TYPE ST_IoT_Communicator :
STRUCT
	{attribute 'iot.DisplayName' := 'Actief Vermogen'}
	{attribute 'iot.Unit' := 'W'}
	{attribute 'iot.ReadOnly' := 'TRUE'}
	{attribute 'iot.DecimalPrecision' := '1'}
	rActiefVermogen	: REAL;
	
	{attribute 'iot.DisplayName' := 'Keuken'}
    bLampKeuken : BOOL;
END_STRUCT
END_TYPE

(* stored: Version 1.1.0.1
   DUT ST_IoT_Communicator: Id {5ae70c63-242c-4cf4-930a-c4e7f109a667} *)
